FUNCTION_BLOCK FB_MasterRobot
VAR
	// flag if slave are connected
	m_slaveOnLine :BOOL :=FALSE;
	m_slaveOnLineCheck :FB_slaveConnectionCheck;
	
	// master-slave motion scale
	m_motionScale :LREAL;
	
	// monitor angle
	m_monitorAngle :LREAL;
	
	// master arm base pose(shoulder pose) in monitor coordinate
	m_shoulderPoseInMonitor :ARRAY[1..2] OF ST_Frame;
	
	// master arms, responsible for arm kinematic and control
	m_masterArms :ARRAY[1..g_mArmNum] OF FB_MasterArm;
	
	// arm state
	m_masterArmState:ARRAY[1..g_mArmNum] OF E_masterArmState:=[E_masterArmState.MasterArmState_Init,E_masterArmState.MasterArmState_Error];
	m_lastMasterArmState:ARRAY[1..g_mArmNum] OF E_masterArmState:=[E_masterArmState.MasterArmState_Init,E_masterArmState.MasterArmState_Error];
	m_nextMasterArmState:ARRAY[1..g_mArmNum] OF E_masterArmState:=[E_masterArmState.MasterArmState_Init,E_masterArmState.MasterArmState_Error];
	
	// index(1 to 4) of slave arm which is tele-linked to master arm
	m_teleSlaveArmIdx:ARRAY[1..g_mArmNum] OF E_MatchedSlaveArmIdx:=[MatchedSlaveArmIdx_NULL, MatchedSlaveArmIdx_null];
	m_matchedMasterArmIdx :ST_MatchedMasterArmIdx;
	m_instruArmState:ARRAY [1..g_mArmNum] OF E_SlaveArmState:=[SlaveArmState_Error, SlaveArmState_Error];
	m_scopeArmState :E_SlaveArmState := SlaveArmState_Error;
	m_scopeArmIndex : E_MatchedSlaveArmIdx :=MatchedSlaveArmIdx_null;
	
	// flag if tele-manipulated slave arm is switched
	m_armSwitchFlag :ARRAY[1..2] OF BOOL := [2(FALSE)];
	
	//master arm selfcheck finshed flag
	m_armSelfCheckFinshedFlag :ARRAY [1..2] OF BOOL;
	
	// flag to enter master-slave control, triggerd by pinching the gripper twice in on second
	m_MSCtrlTriggerFlag :ARRAY[1..g_mArmNum] OF BOOL:=[FALSE, FALSE];
	m_MSCtrlTriggerCheck :ARRAY[1..g_mArmNum] OF FB_MSCtrlTriggerCheck;
	m_MSGripMatchFlag :ARRAY[1..g_mArmNum] OF BOOL:=[FALSE, FALSE];
	m_MSGripMatchCheck :ARRAY[1..g_mArmNum] OF FB_MSGripMatchCheck;
	
	// all arm controller instance 
	m_armCtrlFactory :ARRAY[1..g_mArmNum,1..MasterArmState_totalNum] OF I_MasterArmCtrl;
	m_armError :ARRAY[1..g_mArmNum] OF FB_StateCtrlError;
	m_armInit :ARRAY[1..g_mArmNum] OF FB_StateCtrlInit;
	m_armHome :ARRAY[1..g_mArmNum] OF FB_StateCtrlHome;
	m_armStandBy :ARRAY[1..g_mArmNum] OF FB_StateCtrlStandBy;
	m_armMatching :ARRAY[1..g_mArmNum] OF FB_StateCtrlMatching;
	m_armReady :ARRAY[1..g_mArmNum] OF FB_StateCtrlReady;
	m_armMasterSlave :ARRAY[1..g_mArmNum] OF FB_StateCtrlMasterSlave;
	m_armClutch :ARRAY[1..g_mArmNum] OF FB_StateCtrlClutch;
	m_armEndoscope :ARRAY[1..g_mArmNum] OF FB_StateCtrlEndoscope;
	m_armCart :ARRAY[1..g_mArmNum] OF FB_StateCtrlCart;
	m_armGravityCali :ARRAY[1..g_mArmNum] OF FB_StateCtrlGraCali;
	m_armTest :ARRAY[1..g_mArmNum] OF FB_StateCtrlTest;
	m_armDisable :ARRAY[1..g_mArmNum] OF FB_StateCtrlDisable;
	m_armPerformance :ARRAY[1..g_mArmNum] OF FB_StateCtrlPerformance;
	m_armSelfcheck :ARRAY[1..g_mArmNum] OF FB_StateCtrlSelfcheck;
	m_armPowerOff :ARRAY[1..g_mArmNum] OF FB_StateCtrlPowerOff;	
	m_armGravityBiasCali :ARRAY[1..g_mArmNum] OF FB_StateCtrlGraBiasCali;	
	m_armDynaCali :ARRAY[1..g_mArmNum] OF FB_StateCtrlDynaCali;	
	
	//add code for test
	m_armMotionTest :ARRAY[1..g_mArmNum] OF FB_StateCtrlMotionTest;
	m_armCycleTest :ARRAY[1..g_mArmNum] OF FB_StateCtrlCycleTest;
	m_armFrictionTest :ARRAY[1..g_mArmNum] OF FB_StateCtrlFrictionTest;
	m_armResponseTest :ARRAY[1..g_mArmNum] OF FB_StateCtrlResponseTest;
	m_armDragFreeTest :ARRAY[1..g_mArmNum] OF FB_StateCtrlDragFreeTest;
	m_armManiTest :ARRAY[1..g_mArmNum] OF FB_StateCtrlManiTest;
	m_armCali : ARRAY [1..g_mArmNum] OF FB_StateCtrlArmCali;
	
	// specialized endoscope controller
	m_scopeCtrl :FB_EndoscopeController;
	
	// arm controller interface
	m_armCtrl :ARRAY[1..g_mArmNum] OF I_MasterArmCtrl;
	m_armCtrlCmds :ARRAY[1..g_mArmNum] OF ST_ArmCtrlCmds;
	
	// ultrasonic knife rotation clutch flag
	m_USKnifeRotClutch :ARRAY[1..g_sArmNum] OF BOOL := [4(FALSE)];
	
	// MasterSlave --> (Clutch <----> Endoscope) --> MasterSlave 
	m_masterSlaveFlag :ARRAY[1..g_mArmNum] OF BOOL := [2(FALSE)];
	m_reenterFlag :ARRAY[1..g_mArmNum] OF BOOL;

	m_slavePublicByte : LINT;
END_VAR

 METHOD PROTECTED checkTeleSlaveArmIdx : BOOL
VAR_IN_OUT CONSTANT
	i_masterInputDataPool:ST_MasterInputDataPool;
END_VAR
VAR_STAT
	m_armSwitchR : R_TRIG;
	m_armSwitch : BOOL;
	nextTeleSlaveArmIdx:ARRAY[1..g_mArmNum] OF E_MatchedSlaveArmIdx;
	armDistributionFromUIFlag : BOOL:= FALSE;
END_VAR
nextTeleSlaveArmIdx:=m_teleSlaveArmIdx;
m_armSwitchR(CLK:= i_masterInputDataPool.m_cartStatus.m_armSwitch, Q=> m_armSwitch);
IF m_armSwitch THEN
	m_matchedMasterArmIdx.left1ArmIdx := GVL_interactUI.g_armDistributionInfo.m_leftMappingSlaveArm[1];
	m_matchedMasterArmIdx.left2ArmIdx := GVL_interactUI.g_armDistributionInfo.m_leftMappingSlaveArm[2];
	m_matchedMasterArmIdx.right1ArmIdx := GVL_interactUI.g_armDistributionInfo.m_rightMappingSlaveArm[1];
	m_matchedMasterArmIdx.right2ArmIdx := GVL_interactUI.g_armDistributionInfo.m_rightMappingSlaveArm[2];
END_IF

IF m_matchedMasterArmIdx.left1ArmIdx <> GVL_interactUI.g_armDistributionInfo.m_leftMappingSlaveArm[1] OR m_matchedMasterArmIdx.left2ArmIdx <> GVL_interactUI.g_armDistributionInfo.m_leftMappingSlaveArm[2] THEN
	armDistributionFromUIFlag := TRUE;
END_IF

IF m_matchedMasterArmIdx.left1ArmIdx <=0 OR m_matchedMasterArmIdx.left2ArmIdx <=0 OR m_matchedMasterArmIdx.right1ArmIdx <=0 OR m_matchedMasterArmIdx.right2ArmIdx <=0 THEN
	RETURN;
END_IF

// switch tele-controlled arm index when arm is disenabled
IF i_masterInputDataPool.m_slaveStatus.m_armState[m_matchedMasterArmIdx.left1ArmIdx] = SlaveArmState_Disable THEN
	nextTeleSlaveArmIdx[1]:= m_matchedMasterArmIdx.left2ArmIdx;
ELSIF i_masterInputDataPool.m_slaveStatus.m_armState[m_matchedMasterArmIdx.left2ArmIdx] = SlaveArmState_Disable THEN
	nextTeleSlaveArmIdx[1]:= m_matchedMasterArmIdx.left1ArmIdx;
ELSIF i_masterInputDataPool.m_slaveStatus.m_armState[m_matchedMasterArmIdx.right1ArmIdx] = SlaveArmState_Disable THEN
	nextTeleSlaveArmIdx[2]:= m_matchedMasterArmIdx.right2ArmIdx;
ELSIF i_masterInputDataPool.m_slaveStatus.m_armState[m_matchedMasterArmIdx.right2ArmIdx] = SlaveArmState_Disable THEN
	nextTeleSlaveArmIdx[2]:= m_matchedMasterArmIdx.right1ArmIdx;
END_IF


// switch tele-controlled arm index when endoscope is mounted
IF m_scopeArmIndex = m_matchedMasterArmIdx.left1ArmIdx OR m_scopeArmIndex = m_matchedMasterArmIdx.left2ArmIdx THEN
	// left arm
	IF m_scopeArmIndex = m_matchedMasterArmIdx.left1ArmIdx THEN
		nextTeleSlaveArmIdx[1] := m_matchedMasterArmIdx.left2ArmIdx;
	ELSE
		nextTeleSlaveArmIdx[1] := m_matchedMasterArmIdx.left1ArmIdx;
	END_IF
	
	// right arm
	//check arm have or not trocar
	IF NOT i_masterInputDataPool.m_slaveStatus.m_trocarOnFlag[m_matchedMasterArmIdx.right1ArmIdx] AND m_teleSlaveArmIdx[2] = m_matchedMasterArmIdx.right1ArmIdx
		AND i_masterInputDataPool.m_slaveStatus.m_trocarOnFlag[m_matchedMasterArmIdx.right2ArmIdx]
		AND i_masterInputDataPool.m_slaveStatus.m_armState[m_matchedMasterArmIdx.right2ArmIdx] <> SlaveArmState_Disable THEN
		nextTeleSlaveArmIdx[2] := m_matchedMasterArmIdx.right2ArmIdx;
	ELSIF NOT i_masterInputDataPool.m_slaveStatus.m_trocarOnFlag[m_matchedMasterArmIdx.right2ArmIdx] AND m_teleSlaveArmIdx[2] = m_matchedMasterArmIdx.right2ArmIdx
		AND i_masterInputDataPool.m_slaveStatus.m_trocarOnFlag[m_matchedMasterArmIdx.right1ArmIdx]
		AND i_masterInputDataPool.m_slaveStatus.m_armState[m_matchedMasterArmIdx.right1ArmIdx] <> SlaveArmState_Disable THEN
		nextTeleSlaveArmIdx[2] := m_matchedMasterArmIdx.right1ArmIdx;
	END_IF
	// switch tele-controlled arm index when arm switch is triggerd
	IF m_armSwitch THEN
		IF m_teleSlaveArmIdx[2] = m_matchedMasterArmIdx.right1ArmIdx AND 
						(i_masterInputDataPool.m_slaveStatus.m_armState[m_matchedMasterArmIdx.right2ArmIdx]=SlaveArmState_InstruReady OR i_masterInputDataPool.m_slaveStatus.m_trocarOnFlag[m_matchedMasterArmIdx.right2ArmIdx]) THEN
			nextTeleSlaveArmIdx[2] := m_matchedMasterArmIdx.right2ArmIdx;
		ELSIF 
			m_teleSlaveArmIdx[2]=m_matchedMasterArmIdx.right2ArmIdx AND 
						(i_masterInputDataPool.m_slaveStatus.m_armState[m_matchedMasterArmIdx.right1ArmIdx]=SlaveArmState_InstruReady OR i_masterInputDataPool.m_slaveStatus.m_trocarOnFlag[m_matchedMasterArmIdx.right1ArmIdx]) THEN
			nextTeleSlaveArmIdx[2] := m_matchedMasterArmIdx.right1ArmIdx;
		ELSE
			IF  i_masterInputDataPool.m_slaveStatus.m_armState[m_matchedMasterArmIdx.right1ArmIdx]=SlaveArmState_InstruReady OR i_masterInputDataPool.m_slaveStatus.m_trocarOnFlag[m_matchedMasterArmIdx.right1ArmIdx] THEN
				nextTeleSlaveArmIdx[2] := m_matchedMasterArmIdx.right1ArmIdx;
			ELSIF i_masterInputDataPool.m_slaveStatus.m_armState[m_matchedMasterArmIdx.right2ArmIdx]=SlaveArmState_InstruReady  OR i_masterInputDataPool.m_slaveStatus.m_trocarOnFlag[m_matchedMasterArmIdx.right2ArmIdx] THEN
				nextTeleSlaveArmIdx[2] := m_matchedMasterArmIdx.right2ArmIdx;
			ELSE
				IF armDistributionFromUIFlag THEN
					nextTeleSlaveArmIdx[2] := m_matchedMasterArmIdx.right1ArmIdx;
				END_IF
			END_IF
			
		END_IF
		armDistributionFromUIFlag := FALSE;
	END_IF

ELSIF m_scopeArmIndex = m_matchedMasterArmIdx.right1ArmIdx OR m_scopeArmIndex = m_matchedMasterArmIdx.right2ArmIdx THEN
	// left arm
	//check arm have or not trocar
	IF NOT i_masterInputDataPool.m_slaveStatus.m_trocarOnFlag[m_matchedMasterArmIdx.left1ArmIdx] AND m_teleSlaveArmIdx[1] = m_matchedMasterArmIdx.left1ArmIdx
		AND i_masterInputDataPool.m_slaveStatus.m_trocarOnFlag[m_matchedMasterArmIdx.left2ArmIdx]
		AND i_masterInputDataPool.m_slaveStatus.m_armState[m_matchedMasterArmIdx.left2ArmIdx] <> SlaveArmState_Disable THEN
		nextTeleSlaveArmIdx[1] := m_matchedMasterArmIdx.left2ArmIdx;
	ELSIF NOT i_masterInputDataPool.m_slaveStatus.m_trocarOnFlag[m_matchedMasterArmIdx.left2ArmIdx] AND m_teleSlaveArmIdx[1] = m_matchedMasterArmIdx.left2ArmIdx
		AND i_masterInputDataPool.m_slaveStatus.m_trocarOnFlag[m_matchedMasterArmIdx.left1ArmIdx]
		AND i_masterInputDataPool.m_slaveStatus.m_armState[m_matchedMasterArmIdx.left1ArmIdx] <> SlaveArmState_Disable THEN
		nextTeleSlaveArmIdx[1] := m_matchedMasterArmIdx.left1ArmIdx;
	END_IF
	// switch tele-controlled arm index when arm switch is triggerd
	IF m_armSwitch THEN
		IF m_teleSlaveArmIdx[1]=m_matchedMasterArmIdx.left1ArmIdx AND 
					(i_masterInputDataPool.m_slaveStatus.m_armState[m_matchedMasterArmIdx.left2ArmIdx]=SlaveArmState_InstruReady OR i_masterInputDataPool.m_slaveStatus.m_trocarOnFlag[m_matchedMasterArmIdx.left2ArmIdx]) THEN
			nextTeleSlaveArmIdx[1] := m_matchedMasterArmIdx.left2ArmIdx;
		ELSIF 
			m_teleSlaveArmIdx[1]=m_matchedMasterArmIdx.left2ArmIdx AND 
					(i_masterInputDataPool.m_slaveStatus.m_armState[m_matchedMasterArmIdx.left1ArmIdx]=SlaveArmState_InstruReady OR  i_masterInputDataPool.m_slaveStatus.m_trocarOnFlag[m_matchedMasterArmIdx.left1ArmIdx]) THEN
			nextTeleSlaveArmIdx[1] := m_matchedMasterArmIdx.left1ArmIdx;
		ELSE
			IF  i_masterInputDataPool.m_slaveStatus.m_armState[m_matchedMasterArmIdx.left1ArmIdx]=SlaveArmState_InstruReady OR i_masterInputDataPool.m_slaveStatus.m_trocarOnFlag[m_matchedMasterArmIdx.left1ArmIdx] THEN
				nextTeleSlaveArmIdx[1] := m_matchedMasterArmIdx.left1ArmIdx;
			ELSIF i_masterInputDataPool.m_slaveStatus.m_armState[m_matchedMasterArmIdx.left2ArmIdx]=SlaveArmState_InstruReady OR i_masterInputDataPool.m_slaveStatus.m_trocarOnFlag[m_matchedMasterArmIdx.left2ArmIdx] THEN
				nextTeleSlaveArmIdx[1] := m_matchedMasterArmIdx.left2ArmIdx;
			ELSE
				IF armDistributionFromUIFlag THEN
					nextTeleSlaveArmIdx[1] := m_matchedMasterArmIdx.left1ArmIdx;
				END_IF
			END_IF
		END_IF
		armDistributionFromUIFlag := FALSE;
	END_IF

	// right arm
	IF m_scopeArmIndex = m_matchedMasterArmIdx.right1ArmIdx THEN
		nextTeleSlaveArmIdx[2] := m_matchedMasterArmIdx.right2ArmIdx;
	ELSE
		nextTeleSlaveArmIdx[2] := m_matchedMasterArmIdx.right1ArmIdx;
	END_IF
END_IF

// check if arm-switch is triggerd
m_armSwitchFlag[1]:=m_teleSlaveArmIdx[1] <>  nextTeleSlaveArmIdx[1];
m_armSwitchFlag[2]:=m_teleSlaveArmIdx[2] <>  nextTeleSlaveArmIdx[2];

m_teleSlaveArmIdx:= nextTeleSlaveArmIdx;
END_METHOD

METHOD PROTECTED controllerTransit : BOOL
VAR_INPUT
END_VAR
VAR
	i :INT;
	logStr :STRING;
END_VAR
FOR i:=1 TO g_mArmNum DO 
	IF m_nextMasterArmState[i]<> m_masterArmState[i] THEN
		// reset current controller
		m_armCtrl[i].reset();
		
		// transit to new controller
		m_lastMasterArmState[i]:=m_masterArmState[i];
		m_masterArmState[i]:=m_nextMasterArmState[i];
		m_armCtrl[i]:=m_armCtrlFactory[i,m_masterArmState[i]];
		
		// init next controller
		m_armCtrl[i].Init(m_masterArms[i],m_armCtrlCmds[i]);
		
		// init scope controller
		IF m_masterArmState[i] = MasterArmState_Endoscope  THEN
			m_scopeCtrl.init(m_shoulderPoseInMonitor, m_masterArms, m_armCtrlCmds);
		END_IF
		
		m_masterArms[i].updateCmds(m_armCtrlCmds[i]);
		
		// log
		logStr := 'MasterArm ';
		AGILOG_INFO(logStr, i_printTime:=TRUE, i_lineBreak:=0);
		AGILOG_INFO(i, i_printTime:=FALSE, i_lineBreak:=0);
		logStr := ' Transit To :';
		AGILOG_INFO(logStr, i_printTime:=TRUE, i_lineBreak:=0);
		AGILOG_INFO(m_masterArmState[i], i_printTime:=FALSE, i_lineBreak:=1);
	END_IF
END_FOR
END_METHOD

METHOD PUBLIC getStatus : BOOL
VAR_IN_OUT
	// master robot information, including arm status and cartesian data
	r_masterStatus :ST_MasterStatus;
	
	//master motor in_output to safety check
	r_armMotorData : ST_armMotorData;
	
	// master robot joint data
	r_masterJointsData :ST_MasterJointData;
	
END_VAR

VAR
	i,j:INT;
END_VAR
r_masterStatus.m_motionScale := m_motionScale;
r_masterStatus.m_armState:=m_masterArmState;
r_masterStatus.m_teleSlaveArmIdx := m_teleSlaveArmIdx;
r_masterStatus.m_matchedMasterArmIdx := m_matchedMasterArmIdx;
r_masterStatus.m_masterSlavePoseError := MasterArmControl.m_slaveRobotData.m_masterSlavePoseError;

FOR i:=1 TO g_mArmNum DO
	// current info
	r_masterStatus.m_gripAngle[i]:=m_masterArms[i].gripAngle;
	// cartesion
//	r_masterStatus.m_curArmPose[i]:=m_masterArms[i].curCartPose;
//	r_masterStatus.m_curArmTwist[i]:=m_masterArms[i].curCartTwist;
	r_masterStatus.m_curArmPose[i]:=m_masterArms[i].m_curCartLinkPose;
	r_masterStatus.m_curArmTwist[i]:=m_masterArms[i].m_curCartLinkTwist;
	// joint
	r_masterJointsData.m_curMotorPos[i]:=m_masterArms[i].curMotorPos;
	r_masterJointsData.m_curLinkPos[i]:=m_masterArms[i].curLinkPos;
	r_masterJointsData.m_curJntPos[i]:=m_masterArms[i].curJntPos;
	r_masterJointsData.m_curJntVel[i]:=m_masterArms[i].curJntVel;
	r_masterJointsData.m_curLinkVel[i]:=m_masterArms[i].curLinkVel;
	r_masterJointsData.m_curJntTrq[i]:=m_masterArms[i].curJntTrq;
	r_masterJointsData.m_rawJntCurrent[i]:=m_masterArms[i].rawJntCurrent;
	r_masterJointsData.m_filtJntCurrent[i]:=m_masterArms[i].filtJntCurrent;
	
	// command info
	// cartesion
	r_masterStatus.m_cmdArmPose[i]:=m_masterArms[i].m_cmdCartPose;
	r_masterStatus.m_cmdArmTwist[i]:=m_masterArms[i].m_cmdCartTwist;
	// joint info
	r_masterJointsData.m_cmdJntPos[i]:=m_masterArms[i].m_cmdJntPos;
	r_masterJointsData.m_cmdJntVel[i]:=m_masterArms[i].m_cmdJntVel;
	r_masterJointsData.m_cmdJntTrq[i]:=m_masterArms[i].m_cmdJntTrq;
	r_masterJointsData.m_cmdJntCurrent[i]:=m_masterArms[i].cmdJntCurrent;
	//data to safety check
	r_masterStatus.m_gripHallSensor[i] := m_masterArms[i].m_gripHallSensorIO;
	r_masterStatus.m_slaveHeartBeat := MasterArmControl.m_slaveRobotData.m_heartBeat;
	r_masterStatus.m_IKSuccess[i] := m_armMatching[i].IKSuccess;
	r_masterStatus.m_timePeriod[i] := m_armMatching[i].timePeriod;
	//r_masterStatus.m_selfCheckStatus
	
	//motor data to safety check
	r_armMotorData.m_motorEncSalta[i] :=  m_masterArms[i].motorEncSalta;
	FOR j := 1 TO g_mJntNum DO
		r_armMotorData.m_armMotorInput[i,j] := m_masterArms[i].m_joints[j].m_motorInputs;
		r_armMotorData.m_armMotorOutput[i,j] := m_masterArms[i].m_joints[j].m_motorOutputs;
	END_FOR
	
END_FOR
END_METHOD

METHOD PUBLIC Init : BOOL
VAR_INPUT
END_VAR
VAR
	i:INT;
END_VAR
// init tele-controlled arm index
m_teleSlaveArmIdx[1]:=MatchedSlaveArmIdx_1;
m_teleSlaveArmIdx[2]:=MatchedSlaveArmIdx_3;

// shoulder pose in monitor
m_shoulderPoseInMonitor[1].m_pos[1]:=-g_shoulderDistance/2;
m_shoulderPoseInMonitor[2].m_pos[1]:=g_shoulderDistance/2;

FOR i:=1 TO g_mArmNum DO
	// arm init
	m_masterArms[i].Init(i);
	m_masterArmState[i]:=MasterArmState_Init;
	m_lastMasterArmState[i]:=MasterArmState_Init;
	m_nextMasterArmState[i]:=MasterArmState_Init;
	
	// command init
	m_armCtrlCmds[i].m_jntEnableFlag := g_zeroVec7i;
	m_armCtrlCmds[i].m_jntOPMode := g_allPosMode;
	m_armCtrlCmds[i].m_cmdCartPose := m_masterArms[i].curCartPose;
	m_armCtrlCmds[i].m_cmdCartTwist := g_zeroVec6d;
	m_armCtrlCmds[i].m_cmdJntPos := m_masterArms[i].curJntPos;
	m_armCtrlCmds[i].m_cmdJntVel := g_zeroVec7d;
	m_armCtrlCmds[i].m_cmdJntAcc := g_zeroVec7d;
	m_armCtrlCmds[i].m_cmdJntTrq := g_zeroVec7d;
	
	// generate controller factory
	m_armCtrlFactory[i,MasterArmState_Error] := m_armError[i];
	m_armCtrlFactory[i,MasterArmState_Init] := m_armInit[i];
	m_armCtrlFactory[i,MasterArmState_Home] := m_armHome[i];
	m_armCtrlFactory[i,MasterArmState_Standby] := m_armStandBy[i];
	m_armCtrlFactory[i,MasterArmState_Matching] := m_armMatching[i];
	m_armCtrlFactory[i,MasterArmState_Ready] := m_armReady[i];
	m_armCtrlFactory[i,MasterArmState_MasterSlave] := m_armMasterSlave[i];
	m_armCtrlFactory[i,MasterArmState_Clutch] := m_armClutch[i];
	m_armCtrlFactory[i,MasterArmState_Endoscope] := m_armEndoscope[i];
	m_armCtrlFactory[i,MasterArmState_Cart] := m_armCart[i];
	m_armCtrlFactory[i,MasterArmState_GravityCali] := m_armGravityCali[i];
	m_armCtrlFactory[i,MasterArmState_Test] := m_armTest[i];
	m_armCtrlFactory[i,MasterArmState_Disable] := m_armDisable[i];
	m_armCtrlFactory[i,MasterArmState_Performance] := m_armPerformance[i];
	m_armCtrlFactory[i,MasterArmState_Selfcheck] := m_armSelfcheck[i];
	m_armCtrlFactory[i,MasterArmState_PowerOff] := m_armPowerOff[i];
	m_armCtrlFactory[i,MasterArmState_GravityBiasCali] := m_armGravityBiasCali[i];
	m_armCtrlFactory[i,MasterArmState_masterDynaCali] := m_armDynaCali[i];
	
	
	//add code for test
	//m_armCtrlFactory[i,MasterArmState_Performance] := m_armPerformance[i];
	m_armCtrlFactory[i,MasterArmState_MotionTest] := m_armMotionTest[i];
	m_armCtrlFactory[i,MasterArmState_CycleTest] := m_armCycleTest[i];
	m_armCtrlFactory[i,MasterArmState_FrictionTest] := m_armFrictionTest[i];
	m_armCtrlFactory[i,MasterArmState_ResponseTest] := m_armResponseTest[i];
	m_armCtrlFactory[i,MasterArmState_DragFreeTest] := m_armDragFreeTest[i];
	m_armCtrlFactory[i,MasterArmState_ManiTest] := m_armManiTest[i];
	m_armCtrlFactory[i,MasterArmState_armCali] := m_armCali[i];
	
	// assign controller
	m_armCtrl[i]:=m_armCtrlFactory[i,m_masterArmState[i]];
	m_armCtrl[i].Init(m_masterArms[i],m_armCtrlCmds[i]);
	
	// init master-slave trigger
	m_MSCtrlTriggerCheck[i].init(g_armCtrlCycleTime, 2);
END_FOR
END_METHOD

METHOD PROTECTED MSCtrlTriggerCheck : BOOL
VAR_IN_OUT CONSTANT
		i_masterInputDataPool:ST_MasterInputDataPool;
END_VAR
VAR
	i:INT;
END_VAR
FOR i:=1 TO g_mArmNum DO
	IF MasterArmState_Ready = m_masterArmState[i] AND SlaveArmState_InstruReady = m_instruArmState[i] 
		AND SlaveArmState_ScopeReady = m_scopeArmState AND i_masterInputDataPool.m_cartStatus.m_surgonReady THEN
		m_MSCtrlTriggerFlag[i]:=m_MSCtrlTriggerCheck[i].run(m_masterArms[i]);
	END_IF
	
	IF  MatchedSlaveArmIdx_NULL =  m_teleSlaveArmIdx[i] OR   NOT(i_masterInputDataPool.m_cartStatus.m_surgonReady) 
		OR 	NOT(i_masterInputDataPool.m_slaveStatus.m_instruStauts[m_teleSlaveArmIdx[i]].m_ready) 
		OR m_masterArmState[i] = MasterArmState_Error OR m_masterArmState[i] = MasterArmState_Matching OR i_masterInputDataPool.m_cartStatus.m_consoleInAdjust
		OR  SlaveArmState_Error = m_instruArmState[i] OR SlaveArmState_Disable = m_instruArmState[i]  THEN
		m_MSCtrlTriggerFlag[i]:=FALSE;
		m_MSCtrlTriggerCheck[i].reset();
	END_IF  
END_FOR
END_METHOD

METHOD PROTECTED MSGripMatchCheck : BOOL
VAR_IN_OUT CONSTANT
		i_masterInputDataPool:ST_MasterInputDataPool;
END_VAR
VAR
	i:INT;
	
END_VAR
FOR i:=1 TO g_mArmNum DO
	// grip match check
	IF m_MSCtrlTriggerFlag[i] AND NOT(m_MSGripMatchFlag[i]) THEN
		m_MSGripMatchFlag[i] := m_MSGripMatchCheck[i].run(m_masterArms[i].gripAngle,  i_masterInputDataPool.m_slaveStatus.m_instruStauts[m_teleSlaveArmIdx[i]]);
	END_IF
	
	// reset grip match flag
	IF NOT(m_MSCtrlTriggerFlag[i]) THEN
		m_MSGripMatchFlag[i] := FALSE;
		m_MSGripMatchCheck[i].reset();
	END_IF
	
END_FOR
END_METHOD

METHOD PUBLIC run : BOOL
VAR_IN_OUT CONSTANT
	i_masterInputDataPool:ST_MasterInputDataPool;
END_VAR
VAR
	i:INT;
END_VAR
m_motionScale := i_masterInputDataPool.m_UIData.m_motionScale;
m_monitorAngle := i_masterInputDataPool.m_cartStatus.m_monitorAngle;

// check slave connection
m_slaveOnLine := m_slaveOnLineCheck.check(i_masterInputDataPool.m_slaveStatus.m_slaveHeartBeat);

// update shoulder pose
updateShoulderPose();

// check tele-operated slave arms index
checkTeleSlaveArmIdx(i_masterInputDataPool);

// check if to trig ultrasonic knife ratotation clutch
USKnifeClutchCheck(i_masterInputDataPool);

// update arm status
FOR i:=1 TO g_mArmNum DO
	// update dynamic data
	m_masterArms[i].updateDyna(i_masterInputDataPool.m_masterDynaData);
								
	// update master arm kinematics
	m_masterArms[i].updateStatus();
END_FOR

// state machine transition
stateMachine(i_masterInputDataPool);

// controller transition
controllerTransit();

// run arm controller
FOR i:=1 TO g_mArmNum DO
	// null ptr check
	ASSERT(0 <> m_armCtrl[i]);
	
	// run controller
	m_armCtrl[i].run(m_teleSlaveArmIdx[i], m_shoulderPoseInMonitor[i], m_masterArms[i],
						i_masterInputDataPool.m_slaveStatus,m_armCtrlCmds[i]);
						
	// update commands to drivers
	m_masterArms[i].updateCmds(m_armCtrlCmds[i]);
END_FOR

// run scope controller
IF m_masterArmState[1] = MasterArmState_Endoscope AND m_masterArmState[2] = MasterArmState_Endoscope THEN
	m_scopeCtrl.run(m_teleSlaveArmIdx, m_shoulderPoseInMonitor, m_masterArms, i_masterInputDataPool.m_slaveStatus, m_armCtrlCmds);
	m_masterArms[1].updateCmds(m_armCtrlCmds[1]);
	m_masterArms[2].updateCmds(m_armCtrlCmds[2]);
END_IF
END_METHOD

PROPERTY shoulderPose : ARRAY[1..2] OF ST_Frame
GET
shoulderPose := m_shoulderPoseInMonitor;
END_GET
END_PROPERTY

// state machine check and transit 
METHOD PROTECTED stateMachine : BOOL
VAR_IN_OUT CONSTANT
		i_masterInputDataPool:ST_MasterInputDataPool;
END_VAR
VAR
	i:INT;
	enableClutch :BOOL;
END_VAR
// get instrument arm state
FOR i:=1 TO g_mArmNum DO
	IF MatchedSlaveArmIdx_NULL =  m_teleSlaveArmIdx[i] THEN
		m_instruArmState[i] := SlaveArmState_Error;
	ELSE
		m_instruArmState[i] := i_masterInputDataPool.m_slaveStatus.m_armState[m_teleSlaveArmIdx[i]];
	END_IF
END_FOR

// get endoscope arm state
m_scopeArmState := SlaveArmState_Error;
m_scopeArmIndex := MatchedSlaveArmIdx_null;
FOR i:=1 TO g_sArmNum DO 
	IF InstruType_endoscope =  i_masterInputDataPool.m_slaveStatus.m_instruStauts[i].m_type THEN
		m_scopeArmState := i_masterInputDataPool.m_slaveStatus.m_armState[i];
		m_scopeArmIndex := i;
		EXIT;
	END_IF
END_FOR

// check if master-slave grip angle match
MSCtrlTriggerCheck(i_masterInputDataPool);
MSGripMatchCheck(i_masterInputDataPool);

// State machine transit 
FOR i:=1 TO g_mArmNum DO
	// MasterSlave --> (Clutch <----> Endoscope) --> MasterSlave
	m_masterSlaveFlag[i] := m_masterSlaveFlag[i] AND i_masterInputDataPool.m_cartStatus.m_surgonReady AND NOT(m_armSwitchFlag[i])
						AND (SlaveArmState_MasterSlave =  m_instruArmState[i] OR SlaveArmState_InstruReady =  m_instruArmState[i] OR SlaveArmState_Stop = m_instruArmState[i]);
	m_reenterFlag[i] := m_masterSlaveFlag[i]
					  AND (MasterArmState_Clutch = m_masterArmState[i] OR MasterArmState_Endoscope = m_masterArmState[i] OR MasterArmState_Standby = m_masterArmState[i]
							 OR MasterArmState_Ready = m_masterArmState[i] OR MasterArmState_Matching = m_masterArmState[i])
 					  AND NOT i_masterInputDataPool.m_cartStatus.m_endoscopeSwitch;
	// flag if enable clutch
	enableClutch :=  i_masterInputDataPool.m_cartStatus.m_clutchSwitch OR (m_masterArms[i].handClutchSwitch AND i_masterInputDataPool.m_UIData.m_enableHandClutch);
	
	CASE m_masterArmState[i] OF
		// error
		MasterArmState_Error:
			// to standby
			IF FALSE = i_masterInputDataPool.m_safetyData.m_masterErrFlag[i] THEN
				IF m_armSelfCheckFinshedFlag[i] THEN
					m_nextMasterArmState[i] := MasterArmState_Standby;
				ELSE
					m_nextMasterArmState[i]:=MasterArmState_Home;
				END_IF
			END_IF
			
		// init
		MasterArmState_Init:
			// to home
			IF m_armCtrl[i].isFinished THEN
				// NOTICE: multiple cycles joints back to center during initialization
				// 			need to reset joints encoder data again
				m_masterArms[i].initJntPos();
				m_armSelfCheckFinshedFlag[i] := FALSE;
				m_nextMasterArmState[i]:=MasterArmState_Home;
			END_IF

		//home
		MasterArmState_Home:
			IF m_armCtrl[i].isFinished  THEN
				m_nextMasterArmState[i]:=MasterArmState_GravityBiasCali;
			END_IF
			
		//graivity bias calibration
		MasterArmState_GravityBiasCali:
			IF m_armCtrl[i].isFinished  THEN
				m_armSelfCheckFinshedFlag[i] := TRUE;
				m_nextMasterArmState[i]:=MasterArmState_Standby;
				m_masterArms[i].jntGravityBias := m_armGravityBiasCali[i].m_gravityBias;
			END_IF
		
		//standby
		MasterArmState_Standby:
			// to matching
			IF SlaveArmState_InstruReady = m_instruArmState[i] AND SlaveArmState_ScopeReady = m_scopeArmState 
					AND i_masterInputDataPool.m_slaveStatus.m_slaveAllowInMS AND m_slaveOnLine THEN
				m_nextMasterArmState[i]:=MasterArmState_Matching;
			// to clutch
			ELSIF enableClutch THEN
				m_nextMasterArmState[i] := MasterArmState_Clutch; 
			//to cycle test
			ELSIF g_cycleTest.m_enterCycleTestMode[i] THEN
				m_nextMasterArmState[i] := MasterArmState_CycleTest; 
			// to cart
			ELSIF i_masterInputDataPool.m_cartStatus.m_consoleInAdjust THEN
				m_nextMasterArmState[i] := MasterArmState_Cart;		
			END_IF

		//selfcheck	
		MasterArmState_Selfcheck:
			IF m_armCtrl[i].isFinished  THEN
				m_nextMasterArmState[i]:=MasterArmState_Standby;
			END_IF
		
		//matching
		MasterArmState_Matching:
			// to ready
			IF m_armCtrl[i].isFinished THEN
				m_nextMasterArmState[i]:=MasterArmState_Ready;
			// to clutch
			ELSIF enableClutch THEN
				m_nextMasterArmState[i] := MasterArmState_Clutch; 
			// to standby
			ELSIF SlaveArmState_InstruReady <> m_instruArmState[i] OR SlaveArmState_ScopeReady <> m_scopeArmState
						OR m_armSwitchFlag[i] THEN
				m_nextMasterArmState[i]:=MasterArmState_Standby;
			// to cart
			ELSIF i_masterInputDataPool.m_cartStatus.m_consoleInAdjust THEN
				m_nextMasterArmState[i] := MasterArmState_Cart;
			END_IF
		
		//ready
		MasterArmState_Ready:
			// to standby
			IF SlaveArmState_InstruReady <> m_instruArmState[i] OR SlaveArmState_ScopeReady <> m_scopeArmState
					OR m_armSwitchFlag[i] THEN
				m_nextMasterArmState[i]:=MasterArmState_Standby;
			// to clutch
			ELSIF enableClutch THEN
				m_nextMasterArmState[i] := MasterArmState_Clutch; 
			// to cart
			ELSIF i_masterInputDataPool.m_cartStatus.m_consoleInAdjust THEN
				m_nextMasterArmState[i] := MasterArmState_Cart;
			// to master-slave
			ELSIF SlaveArmState_InstruReady = m_instruArmState[i] AND SlaveArmState_ScopeReady = m_scopeArmState AND i_masterInputDataPool.m_cartStatus.m_surgonReady 
					AND ((m_MSCtrlTriggerFlag[i] AND m_MSGripMatchFlag[i]) OR m_reenterFlag[i])AND NOT(i_masterInputDataPool.m_cartStatus.m_consoleInAdjust)  
					AND (NOT i_masterInputDataPool.m_cartStatus.m_endoscopeSwitch OR i_masterInputDataPool.m_UIData.m_masterArmDisableFlag[1] OR i_masterInputDataPool.m_UIData.m_masterArmDisableFlag[2])THEN
				m_nextMasterArmState[i] := MasterArmState_MasterSlave;
			// to standby
			ELSIF NOT i_masterInputDataPool.m_slaveStatus.m_slaveAllowInMS OR NOT m_slaveOnLine THEN
				m_nextMasterArmState[i]:=MasterArmState_Standby;
			//to cycle test
			ELSIF g_cycleTest.m_enterCycleTestMode[i] THEN
				m_nextMasterArmState[i] := MasterArmState_CycleTest; 	
			
			END_IF
		
		//MasterSlave
		MasterArmState_MasterSlave:
			IF (g_motionTest.m_MSPrecisionTest[i]=FALSE)THEN			
				// to standdy
				IF  (SlaveArmState_InstruReady <> m_instruArmState[i] AND SlaveArmState_MasterSlave <> m_instruArmState[i] AND SlaveArmState_Stop <> m_instruArmState[i])
					OR (SlaveArmState_ScopeReady <> m_scopeArmState AND SlaveArmState_Stop <> m_scopeArmState AND SlaveArmState_EndoScope <> m_scopeArmState)
					OR NOT(i_masterInputDataPool.m_cartStatus.m_surgonReady) OR m_armSwitchFlag[i] 
					OR (i_masterInputDataPool.m_cartStatus.m_endoscopeSwitch AND ((NOT i_masterInputDataPool.m_UIData.m_masterArmDisableFlag[1])AND (NOT i_masterInputDataPool.m_UIData.m_masterArmDisableFlag[2])) )THEN
					m_nextMasterArmState[i]:=MasterArmState_Standby;
				// to clutch
				ELSIF enableClutch THEN
					m_nextMasterArmState[i] := MasterArmState_Clutch; 
				//to standby
				ELSIF NOT m_slaveOnLine THEN
					m_nextMasterArmState[i] := MasterArmState_Standby;
				// to match
				ELSIF NOT(m_armMasterSlave[i].initRotErrCheck) THEN
					m_nextMasterArmState[i]:=MasterArmState_Matching;
				ELSE
					m_masterSlaveFlag[i] := TRUE;
				END_IF		
			ELSE
								
				// to standdy
				IF  (SlaveArmState_InstruReady <> m_instruArmState[i] AND SlaveArmState_MasterSlave <> m_instruArmState[i])
					OR SlaveArmState_ScopeReady <> m_scopeArmState OR m_armSwitchFlag[i] THEN
					m_nextMasterArmState[i]:=MasterArmState_Standby;
				// to clutch
				ELSIF enableClutch THEN
					m_nextMasterArmState[i] := MasterArmState_Clutch; 
				//to standby
				ELSIF NOT m_slaveOnLine THEN
					m_nextMasterArmState[i] := MasterArmState_Standby;
				END_IF				
			END_IF
			
		//Clutch
		MasterArmState_Clutch:
			IF NOT(enableClutch) THEN
				// to master slave 
				IF (m_lastMasterArmState[i] = MasterArmState_MasterSlave OR m_masterSlaveFlag[i])  THEN
					m_nextMasterArmState[i] := MasterArmState_MasterSlave;
				// to standby
				ELSE
					m_nextMasterArmState[i]:=MasterArmState_Standby;
				END_IF
			END_IF
		
		// Endoscope 
		MasterArmState_Endoscope:
			IF NOT(i_masterInputDataPool.m_cartStatus.m_endoscopeSwitch) THEN
				// to master slave 
				IF m_lastMasterArmState[i] = MasterArmState_MasterSlave OR m_masterSlaveFlag[i] THEN
					m_nextMasterArmState[i] := MasterArmState_MasterSlave;
				// to standby
				ELSE
					m_nextMasterArmState[i]:=MasterArmState_Standby;
				END_IF
			// to standby
			ELSIF NOT(i_masterInputDataPool.m_cartStatus.m_surgonReady) 
				OR MasterArmState_Endoscope<> m_masterArmState[1] OR MasterArmState_Endoscope<> m_masterArmState[2]
				OR (SlaveArmState_ScopeReady <> m_scopeArmState AND SlaveArmState_EndoScope <> m_scopeArmState) THEN
				m_nextMasterArmState[i] := MasterArmState_Standby;
			// to clutch
			ELSIF enableClutch THEN
				m_nextMasterArmState[i] := MasterArmState_Clutch; 
			// to cart
			ELSIF i_masterInputDataPool.m_cartStatus.m_consoleInAdjust THEN
				m_nextMasterArmState[i] := MasterArmState_Cart;
			//to standby
			ELSIF NOT m_slaveOnLine THEN
				m_nextMasterArmState[i] := MasterArmState_Standby;
			END_IF
			
		// Cart 
		MasterArmState_Cart:
			// to standby
			IF NOT( i_masterInputDataPool.m_cartStatus.m_consoleInAdjust) THEN
				m_nextMasterArmState[i] := MasterArmState_Standby;
			END_IF
		
		//Gravity Calibration
		MasterArmState_GravityCali:
			// to standby
			IF  m_armCtrl[i].isFinished THEN
				m_nextMasterArmState[i]:=MasterArmState_Standby;
			END_IF
	
		//arm test
		MasterArmState_Test:
			// to standby
			IF  m_armCtrl[i].isFinished THEN
				m_nextMasterArmState[i]:=MasterArmState_Standby;
			END_IF
			
		//arm Performance
		MasterArmState_Performance:
			// to standby
			IF  m_armCtrl[i].isFinished THEN
				m_nextMasterArmState[i]:=MasterArmState_Standby;
			END_IF
			
		//arm disable
		MasterArmState_Disable:
			// to init
			IF  NOT(i_masterInputDataPool.m_UIData.m_masterArmDisableFlag[i]) THEN
				m_armSelfCheckFinshedFlag[i] := FALSE;
				m_nextMasterArmState[i]:=MasterArmState_Init;
			END_IF
			
		// dynamic calibration
		MasterArmState_masterDynaCali:	
			IF m_armCtrl[i].isFinished THEN
				m_nextMasterArmState[i] :=MasterArmState_Standby;
			END_IF
			
		MasterArmState_CycleTest:
			IF m_armCtrl[i].isFinished OR NOT g_cycleTest.m_enterCycleTestMode[i] THEN
				m_nextMasterArmState[i] :=MasterArmState_Standby;
			END_IF
	END_CASE
	
	
	// to precision test
	IF (g_motionTest.m_enterPrecisionTestMode[i]=TRUE) AND NOT(m_masterArmState[i]=MasterArmState_MotionTest) THEN
		m_nextMasterArmState[i] := MasterArmState_MotionTest;
	END_IF
	//precision exit
	IF (g_motionTest.m_enterPrecisionTestMode[i]=FALSE) AND (m_masterArmState[i]=MasterArmState_MotionTest) THEN
		m_nextMasterArmState[i] := MasterArmState_Standby;
	END_IF	
	
	// to MS precision test
	IF (g_motionTest.m_MSPrecisionTest[i]=TRUE) AND NOT(m_masterArmState[i]=MasterArmState_MasterSlave) THEN
		//m_nextMasterArmState[i] := MasterArmState_MasterSlave;
	END_IF
	
	// to MS precision test
	IF (g_motionTest.m_MSPrecisionTest[i]=TRUE) AND NOT(m_masterArmState[i]=MasterArmState_MasterSlave) THEN
		IF (m_masterArmState[i]=MasterArmState_Ready) THEN
			IF SlaveArmState_InstruReady = m_instruArmState[i] AND SlaveArmState_ScopeReady = m_scopeArmState AND NOT(i_masterInputDataPool.m_cartStatus.m_consoleInAdjust) THEN
				m_nextMasterArmState[i] := MasterArmState_MasterSlave;
			END_IF
		END_IF		
	END_IF	
	
	// to MasterArmState_TestCycle
	//IF (g_cycleTest.m_enterCycleTestMode[i] OR g_cycleTest.m_enterESDTest[i]) AND NOT(m_masterArmState[i]=MasterArmState_CycleTest) THEN
	//	m_nextMasterArmState[i] := MasterArmState_CycleTest;
	//END_IF
	
	//MasterArmState_TestCycle exit
	//IF (g_cycleTest.m_enterCycleTestMode[i]=FALSE) AND (g_cycleTest.m_enterESDTest[i]=FALSE) AND(m_masterArmState[i]=MasterArmState_CycleTest) THEN
	//	m_nextMasterArmState[i] := MasterArmState_Standby;
	//END_IF
	
	// to MasterArmState_TestFriction
	IF (g_frictionTest.m_testMode[i]=TRUE) AND NOT(m_masterArmState[i]=MasterArmState_FrictionTest) THEN
		m_nextMasterArmState[i] := MasterArmState_FrictionTest;
	END_IF
	
	// MasterArmState_TestFriction exit
	IF (g_frictionTest.m_testMode[i]=FALSE) AND (m_MasterArmState[i]=MasterArmState_FrictionTest) THEN
		m_nextMasterArmState[i] := MasterArmState_Standby;
	END_IF
	
	// to MasterArmState_TestDragFree
	IF (g_frictionTest.m_clutchMode[i]=TRUE) AND (m_masterArms[i].handClutchSwitch=TRUE) AND NOT(m_masterArmState[i]=MasterArmState_DragFreeTest) THEN
		m_nextMasterArmState[i] := MasterArmState_DragFreeTest;
	END_IF
	
	// MasterArmState_TestDragFree exit
	IF (m_masterArms[i].handClutchSwitch=FALSE) AND (m_MasterArmState[i]=MasterArmState_DragFreeTest) THEN
		m_nextMasterArmState[i] := MasterArmState_Standby;
	END_IF
	
	// to home
	IF (g_frictionTest.m_getHome[i]=TRUE) AND NOT(m_masterArmState[i]=MasterArmState_Home) THEN
		m_nextMasterArmState[i] := MasterArmState_Home;
	END_IF
	
	//MasterArmState_TestMani
	IF (g_maniTest.m_testStart[i]=TRUE) AND NOT(m_masterArmState[i]=MasterArmState_ManiTest) THEN
		m_nextMasterArmState[i]:=MasterArmState_ManiTest;
	END_IF
	
	//MasterArmState_TestMani exit
	IF (g_maniTest.m_testStart[i]=FALSE) AND (m_masterArmState[i]=MasterArmState_ManiTest) THEN
		m_nextMasterArmState[i]:=MasterArmState_Standby;
	END_IF
	
	//robot calibration 
	IF GVL_armCali.g_armEnterCaliMode[i] AND (m_masterArmState[i]<=MasterArmState_Standby) THEN
		m_nextMasterArmState[i] := MasterArmState_armCali;
	ELSIF NOT GVL_armCali.g_armEnterCaliMode[i] AND (m_masterArmState[i]=MasterArmState_armCali) THEN
		m_nextMasterArmState[i] := MasterArmState_Init;
	END_IF	
	
	//fault mask
	IF (g_specialSignal.m_faultMask[i]) THEN
		CONTINUE;
	END_IF
	
	
	
	
	// arm disable
	IF i_masterInputDataPool.m_UIData.m_masterArmDisableFlag[i] THEN
		m_nextMasterArmState[i] := MasterArmState_Disable;
	// error check
	ELSIF i_masterInputDataPool.m_safetyData.m_masterErrFlag[i] THEN
		m_nextMasterArmState[i] := MasterArmState_Error;
	//to poweroff
	ELSIF  GVL_interactUI.g_uiPowerOffEnable	THEN
		m_nextMasterArmState[i] := MasterArmState_PowerOff;		
	END_IF
	
END_FOR

// To Endoscope Control 
IF SlaveArmState_ScopeReady = m_scopeArmState AND i_masterInputDataPool.m_cartStatus.m_endoscopeSwitch AND i_masterInputDataPool.m_cartStatus.m_surgonReady AND
  (MasterArmState_Standby = m_masterArmState[1] OR MasterArmState_Ready = m_masterArmState[1] OR MasterArmState_MasterSlave = m_masterArmState[1]) AND 
  (MasterArmState_Standby = m_masterArmState[2] OR MasterArmState_Ready = m_masterArmState[2] OR MasterArmState_MasterSlave = m_masterArmState[2]) 
	AND i_masterInputDataPool.m_slaveStatus.m_slaveAllowInMS THEN
		m_nextMasterArmState[1] := MasterArmState_Endoscope;
		m_nextMasterArmState[2] := MasterArmState_Endoscope;

END_IF
END_METHOD

METHOD PROTECTED updateShoulderPose : BOOL
VAR_INPUT
END_VAR
VAR
	monitorRot :mat3d;
END_VAR
// base monitor frame(0 rotation angle) in current monitor frame 
monitorRot := rotY( -m_monitorAngle);

// shoulder pose in current monitor frame
matMultiply(g_shoulderRotInMonitor,monitorRot, m_shoulderPoseInMonitor[1].m_rot);
m_shoulderPoseInMonitor[2].m_rot:=m_shoulderPoseInMonitor[1].m_rot;
END_METHOD

METHOD USKnifeClutchCheck : BOOL
VAR_IN_OUT CONSTANT
	i_masterInputDataPool:ST_MasterInputDataPool;
END_VAR

VAR
	i:INT;
END_VAR
FOR i:=1 TO g_sArmNum DO
	IF NOT(i_masterInputDataPool.m_slaveStatus.m_instruStauts[i].m_ready) THEN
		m_USKnifeRotClutch[i] := FALSE;
	END_IF
END_FOR

FOR i:=1 TO g_mArmNum DO
	IF (i_masterInputDataPool.m_slaveStatus.m_instruStauts[m_teleSlaveArmIdx[i]].m_type = InstruType_UltrasoundKnifeS OR i_masterInputDataPool.m_slaveStatus.m_instruStauts[m_teleSlaveArmIdx[i]].m_type = InstruType_UltrasoundKnifeU)
		AND  m_masterArmState[i] = MasterArmState_Clutch AND m_masterArms[i].handClutchSwitch THEN
		m_USKnifeRotClutch[m_teleSlaveArmIdx[i]] := TRUE;
	END_IF
END_FOR
END_METHOD

END_FUNCTION_BLOCK

(* stored: Version 1.1.0.1, ProductVersion 3.1.4024.11
   POU FB_MasterRobot: Id {8cbdb2ba-9735-46e3-8cbc-296330acc8cc}, SpecialFunc None
   Folder property: Id {8f86633f-3f94-408a-ac9b-8ee0ebd6bdac}
   Method checkTeleSlaveArmIdx: Id {e877542b-f696-4449-b007-3e9fbc5ffaab}
   Method controllerTransit: Id {43db9dd9-8e13-4a66-a84f-800b29862df6}
   Method getStatus: Id {b6139e8c-2703-424c-9761-ad1add6b1ff1}
   Method Init: Id {610a17f3-34c5-4e3c-bbbc-19f9c2f46946}
   Method MSCtrlTriggerCheck: Id {848392d9-479b-4441-b2d2-6aff07409695}
   Method MSGripMatchCheck: Id {304edd15-5d78-42c9-ab19-2d8f9909a033}
   Method run: Id {ed6f787a-4dc0-4602-b386-92a3c3880a23}
   Property shoulderPose: Id {6004f8dc-7ada-4ad2-9d1e-93605d16d31e}
   Get Get: Id {4fa3cfe8-ad39-4a7f-9fe0-f47bb30c0cd4}
   Method stateMachine: Id {b9cc8560-9309-49e3-93b5-28cb02b4f5cc}
   Method updateShoulderPose: Id {fb1a54a0-df1a-4720-ac59-3d297fc90e27}
   Method USKnifeClutchCheck: Id {99618810-c3d1-4d48-8924-a195c5080579} *)
